// TIA Portal V17 export
FUNCTION "多网络示例" : Void   // FC, LAD
{ S7_Optimized_Access := 'TRUE' }
VERSION : 0.1
// stored: AutoNumber true, IsIECCheckEnabled false, SetENOAutomatically false
BEGIN

REGION Network 1
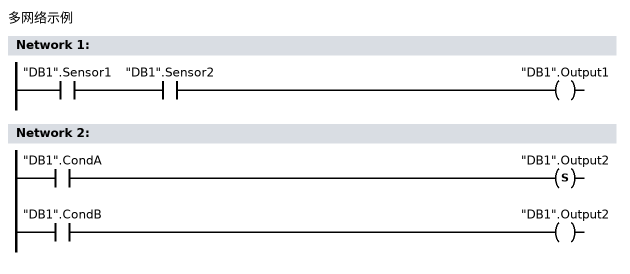
   RUNG wire#powerrail
      Contact( "DB1".Sensor1 )
      Contact( "DB1".Sensor2 )
      Coil( "DB1".Output1 )
   END_RUNG
   // the same network as SCL:
   "DB1".Output1 := "DB1".Sensor1 AND "DB1".Sensor2;
END_REGION

REGION Network 2
   RUNG wire#powerrail
      Contact( "DB1".CondA )
      S_Coil( "DB1".Output2 )
   END_RUNG
   RUNG wire#powerrail
      Contact( "DB1".CondB )
      Coil( "DB1".Output2 )
   END_RUNG
   // the same network as SCL:
   IF "DB1".CondA THEN "DB1".Output2 := TRUE; END_IF;
   "DB1".Output2 := "DB1".CondB;
END_REGION
END_FUNCTION
